TYPE stHIBOTLocalPara :
STRUCT
 	stClampPara  :  stRealPara;//夹持
	stRotateClampPara :  stRealPara;//旋转
	stRotateRelAngle:REAL;//相对旋转角度
END_STRUCT
END_TYPE

(* stored: Version 1.1.0.1, ProductVersion 3.1.4024.9
   DUT stHIBOTLocalPara: Id {45708503-8cfa-4206-952a-1a8c90ce5179} *)
